DATA_BLOCK DB 87
TITLE =
VERSION : 0.0

 FB 87
BEGIN

modes.WKM1PROC.batchCycle := TRUE;
modes.WKM1PROC.autoSwitch := TRUE;
pilot.pilot_F1.F1TurM1ACT.highSpeedPB := TRUE;

END_DATA_BLOCK